TYPE Udt_PlantControl_Mode_2 :
STRUCT
	Startet_Out : BOOL;
	Stopped_Out : BOOL;
	Reset_Out : BOOL;
END_STRUCT
END_TYPE

(* stored: Version 1.1.0.1, ProductVersion 3.1.4024.13
   DUT Udt_PlantControl_Mode_2: Id {7375d448-a3e6-4fef-8c3a-42f1227426f1} *)
